// TIA Portal V16 export
// export: Created 2021-04-06T19:52:18.9493995Z, ExportSetting WithDefaults, DisplayName Totally Integrated Automation Portal, DisplayVersion V16, DisplayName TIA Portal Version Control Interface, DisplayVersion V16, DisplayName TIA Portal Openness, DisplayVersion V16, DisplayName STEP 7 Professional, DisplayVersion V16, DisplayName STEP 7 Safety, DisplayVersion V16, DisplayName WinCC Unified SCADA Engineering System, DisplayVersion V16
TYPE "cleaningMode"
// stored: IsFailsafeCompliant false
   STRUCT
      allWeightModuleReady : Bool;   // Все весоизмерительные модули готовы
      pauseClean : Bool;   // пауза очистки
      progressClean : Int;   // прогресс очистки
      runClean : Bool;   // запуск очистки
      timeClean : Int;   // время очистки
   END_STRUCT;
END_TYPE
